Omron CX-Programmer project NewProject (CX-Programmer 9.61)

# PLC Module_3_PIDAT: CP1H XA

## Global symbols (name address type ; comment)
100.00 BOOL  ; 100.00 - PUMP
100.01 BOOL  ; 100.01 - SV1
100.02 BOOL  ; 100.03 - SV2
100.03 BOOL  ; 100.03 - SV3
202 CHANNEL  ; Float Level Sensor Input
210 CHANNEL  ; Servo Valve Output Control
D1 CHANNEL  ; Screen Display
D10 CHANNEL  ; SCADA - C - SV
D100 CHANNEL  ; C - Set Point Value
D101 CHANNEL  ; C+1 - P Value
D102 CHANNEL  ; C+2 - I Value
D103 CHANNEL  ; C+3 - D Value
D104 CHANNEL  ; C+4 - Sampling Period
D105 CHANNEL  ; C+5 - PID Settings Designation
D106 CHANNEL  ; C+6 - MV Control
D107 CHANNEL  ; C+7 - MV Min. Value
D108 CHANNEL  ; C+8 - MV Max. Value
D109 CHANNEL  ; C+9 - Auto Tuning Settings
D11 CHANNEL  ; GUI - C+1 - P Value
D110 CHANNEL  ; C+10 - Limit-Cycle Hysteresis
D12 CHANNEL  ; GUI - C+2 - I Value
D13 CHANNEL  ; GUI - C+3 - D Value
D14 CHANNEL  ; GUI - C+4 - Sampling Period
D20 CHANNEL  ; Linear Function Offset
D21 CHANNEL  ; Delta Input Range
D22 CHANNEL  ; Delta Output Range
D23 CHANNEL  ; Max. Output
D24 CHANNEL  ; Min. Output
D27 CHANNEL  ; User Input Password
D28 CHANNEL  ; Correct Password
D30 CHANNEL  ; Min. Output
D31 CHANNEL  ; Min. Input
D32 CHANNEL  ; Max. Output
D33 CHANNEL  ; Max. Input
D35 CHANNEL  ; Min. Output
D36 CHANNEL  ; Min. Input
D37 CHANNEL  ; Max. Output
D38 CHANNEL  ; Max. Input
D40 CHANNEL  ; Tank Water Level BCD Equivalent
D41 CHANNEL  ; Set Point Level BCD Equivalent
D42 CHANNEL  ; Current Supplied to Servo Valve (mA)
D5 CHANNEL  ; User Input Password
D6 CHANNEL  ; Correct Password
T0000 BOOL  ; Initialization Delay
T0001 BOOL  ; Autotuning Delay
T0002 BOOL  ; Password Screen Shift Delay

## Program Tank_Water_Control_by_PIDAT (cyclic task 0)
Local symbols
PUMP 10.00 BOOL  ; 10.00 - PUMP
START 7.00 BOOL  ; 7.00 - START
SV1 11.00 BOOL  ; 11.00 - SV1
SV2 12.00 BOOL  ; 12.00 - SV2
SV3 13.00 BOOL  ; 13.00 - SV3

### Section Initialization_Section

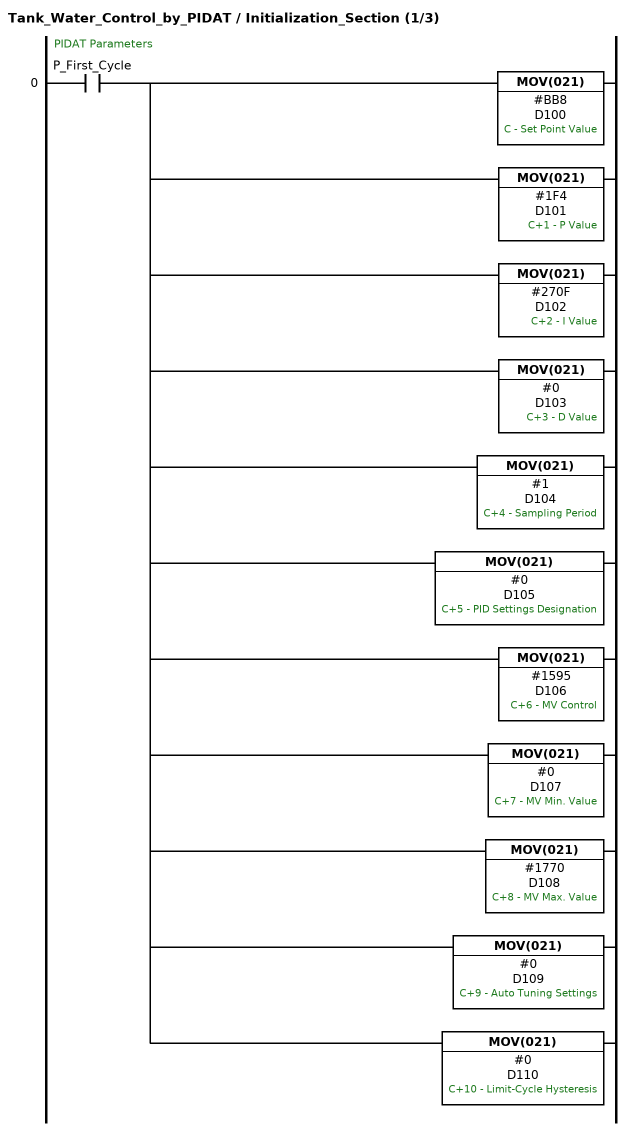
; rung 0: PIDAT Parameters
LD P_First_Cycle
MOV(021) #BB8 D100  ; C - Set Point Value
MOV(021) #1F4 D101  ; C+1 - P Value
MOV(021) #270F D102  ; C+2 - I Value
MOV(021) #0 D103  ; C+3 - D Value
MOV(021) #1 D104  ; C+4 - Sampling Period
MOV(021) #0 D105  ; C+5 - PID Settings Designation
MOV(021) #1595 D106  ; C+6 - MV Control
MOV(021) #0 D107  ; C+7 - MV Min. Value
MOV(021) #1770 D108  ; C+8 - MV Max. Value
MOV(021) #0 D109  ; C+9 - Auto Tuning Settings
MOV(021) #0 D110  ; C+10 - Limit-Cycle Hysteresis

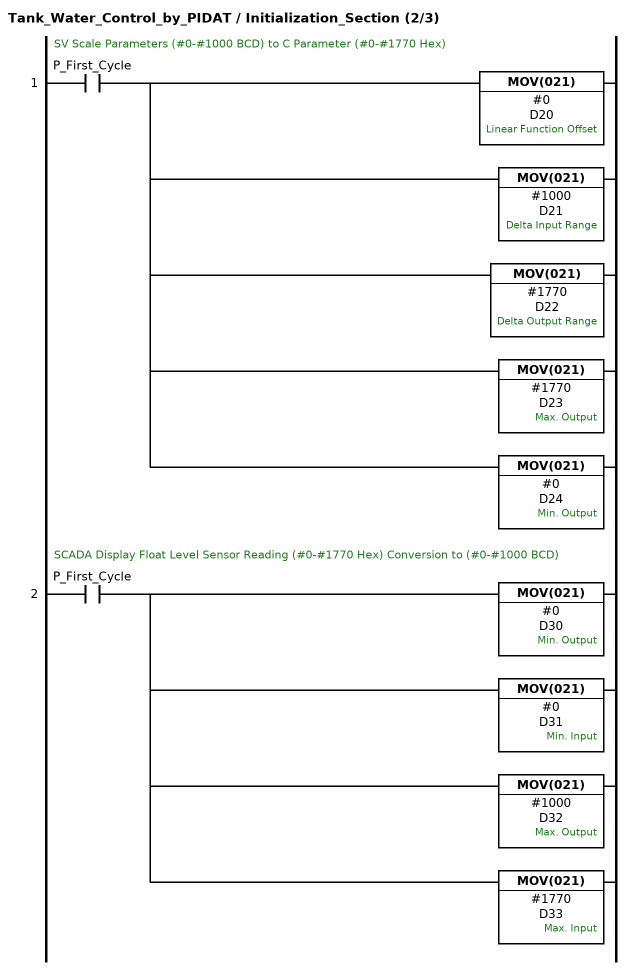
; rung 1: SV Scale Parameters (#0-#1000 BCD) to C Parameter (#0-#1770 Hex)
LD P_First_Cycle
MOV(021) #0 D20  ; Linear Function Offset
MOV(021) #1000 D21  ; Delta Input Range
MOV(021) #1770 D22  ; Delta Output Range
MOV(021) #1770 D23  ; Max. Output
MOV(021) #0 D24  ; Min. Output
; rung 2: SCADA Display Float Level Sensor Reading (#0-#1770 Hex) Conversion to (#0-#1000 BCD)
LD P_First_Cycle
MOV(021) #0 D30  ; Min. Output
MOV(021) #0 D31  ; Min. Input
MOV(021) #1000 D32  ; Max. Output
MOV(021) #1770 D33  ; Max. Input

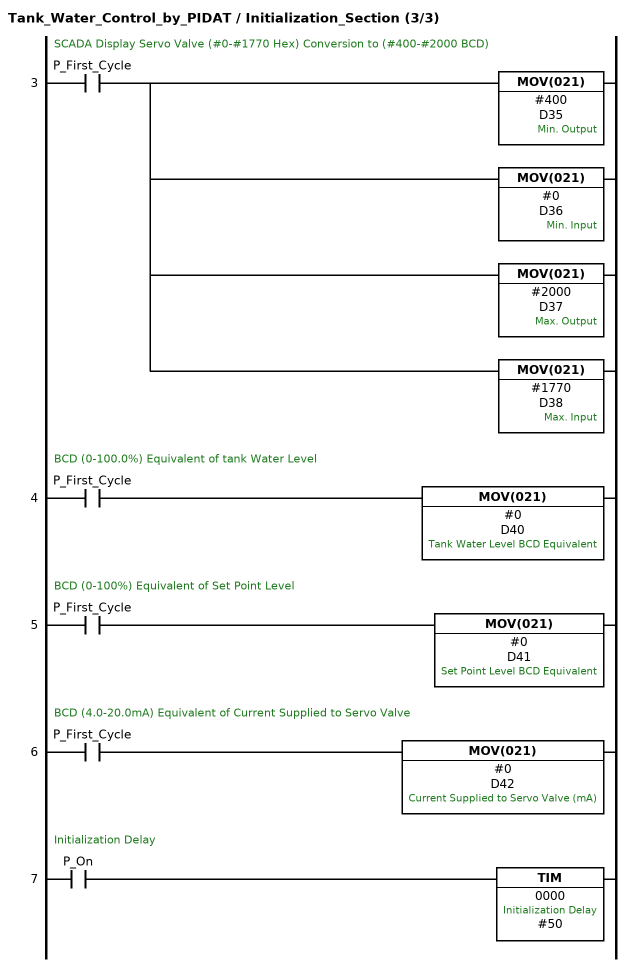
; rung 3: SCADA Display Servo Valve (#0-#1770 Hex) Conversion to (#400-#2000 BCD)
LD P_First_Cycle
MOV(021) #400 D35  ; Min. Output
MOV(021) #0 D36  ; Min. Input
MOV(021) #2000 D37  ; Max. Output
MOV(021) #1770 D38  ; Max. Input
; rung 4: BCD (0-100.0%) Equivalent of tank Water Level
LD P_First_Cycle
MOV(021) #0 D40  ; Tank Water Level BCD Equivalent
; rung 5: BCD (0-100%) Equivalent of Set Point Level
LD P_First_Cycle
MOV(021) #0 D41  ; Set Point Level BCD Equivalent
; rung 6: BCD (4.0-20.0mA) Equivalent of Current Supplied to Servo Valve
LD P_First_Cycle
MOV(021) #0 D42  ; Current Supplied to Servo Valve (mA)
; rung 7: Initialization Delay
LD P_On
TIM 0000 #50  ; Initialization Delay

### Section Main_Program_Section

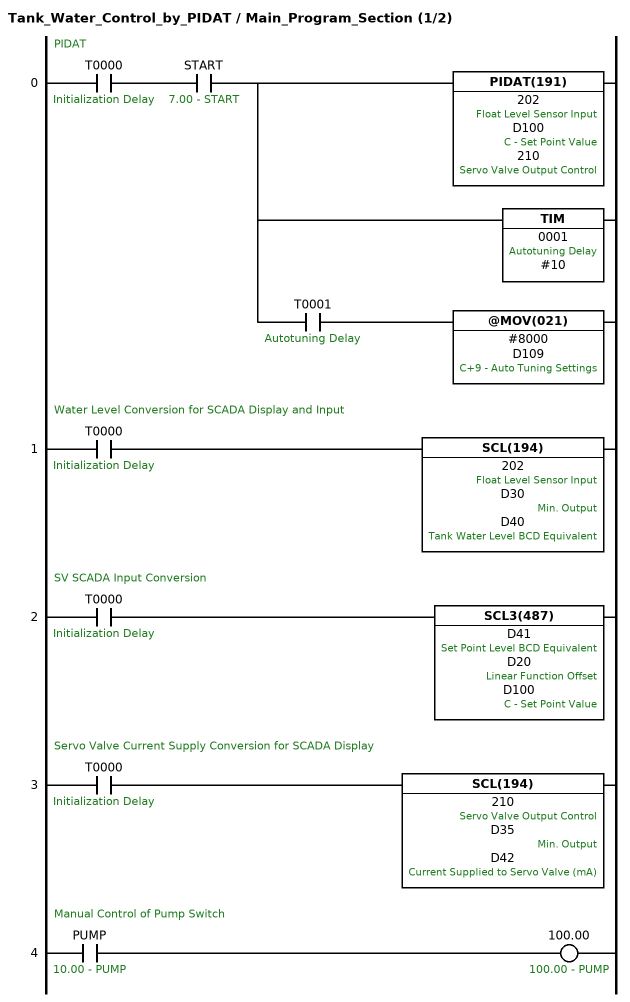
; rung 0: PIDAT
LD T0000  ; Initialization Delay
AND START  ; 7.00 - START
PIDAT(191) 202 D100 210  ; Float Level Sensor Input, C - Set Point Value, Servo Valve Output Control
TIM 0001 #10  ; Autotuning Delay
AND T0001  ; Autotuning Delay
@MOV(021) #8000 D109  ; C+9 - Auto Tuning Settings
; rung 1: Water Level Conversion for SCADA Display and Input
LD T0000  ; Initialization Delay
SCL(194) 202 D30 D40  ; Float Level Sensor Input, Min. Output, Tank Water Level BCD Equivalent
; rung 2: SV SCADA Input Conversion
LD T0000  ; Initialization Delay
SCL3(487) D41 D20 D100  ; Set Point Level BCD Equivalent, Linear Function Offset, C - Set Point Value
; rung 3: Servo Valve Current Supply Conversion for SCADA Display
LD T0000  ; Initialization Delay
SCL(194) 210 D35 D42  ; Servo Valve Output Control, Min. Output, Current Supplied to Servo Valve (mA)
; rung 4: Manual Control of Pump Switch
LD PUMP  ; 10.00 - PUMP
OUT 100.00  ; 100.00 - PUMP

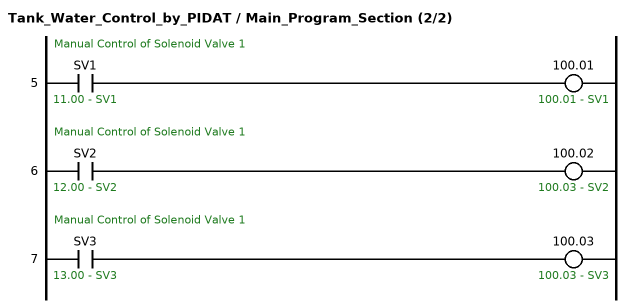
; rung 5: Manual Control of Solenoid Valve 1
LD SV1  ; 11.00 - SV1
OUT 100.01  ; 100.01 - SV1
; rung 6: Manual Control of Solenoid Valve 1
LD SV2  ; 12.00 - SV2
OUT 100.02  ; 100.03 - SV2
; rung 7: Manual Control of Solenoid Valve 1
LD SV3  ; 13.00 - SV3
OUT 100.03  ; 100.03 - SV3

### Section END
; rung 0
END(001)